(* IEC 61131-3 sources: Industry-PLC-LLM/data/PLCBEAD_repo/PLCBEAD_PLCEmbed-main/PLC-BEAD/Source/GEB/_BYTE_TO_DINT, 1 file *)

(* ---- _BYTE_TO_DINT.ST ---- *)
FUNCTION _BYTE_TO_DINT:DINT
	VAR_INPUT
		IN :	BYTE;
	END_VAR

	_BYTE_TO_DINT := USINT_TO_DINT(BYTE_TO_USINT(IN));
END_FUNCTION

PROGRAM program0
  VAR
    LocalVar0 : BYTE;
	LocalOUT  : DINT;
  END_VAR

  LocalOUT := _BYTE_TO_DINT(LocalVar0);
END_PROGRAM
